Universal Robots PolyScope program: pr1.urp

Program pr1 (installation=default directory=/programs createdIn=5.5.1.82186 lastSavedIn=5.5.1.82186 robotSerialNumber=20195300809)
Calibrated DH parameters: a=[-0.000085, -0.20076, -0.212369, 0.000121, -0.000118, 0]; d=[0.15185, -26.306375, 24.753047, 1.684739, 0.085386, 0.092088]; alpha=[1.572149, -0.00522, -0.011864, 1.571339, -1.571085, 0]; deltaTheta=[0, 0.599885, -0.513355, -0.086555, 0.000006, 0]
BeforeStart
  URCap Gripper (Robotiq_Grippers, Robotiq Inc.) dataModel(position=0.0, force=100.0, speed=100.0, positionInDouble=0.0, forceInDouble=100.0, speedInDouble=100.0, slaveIds=[9], blocking=true)
  MoveJ speed 30 deg/s, acceleration 80 deg/s^2 (useActiveTCP=true) feature=Base
    Waypoint punt1: TCP in base x=-102.832 y=-139.085 z=685.946 mm, rx=-1.1427 ry=-1.3106 rz=1.2216 rad; joints [-11.105, -100.438, 18.426, -96.643, -75.028, -3.585] deg
Robot Program (runOnlyOnce=false)
  MoveJ speed 15 deg/s, acceleration 80 deg/s^2 (useActiveTCP=true) feature=Base
    Waypoint Agafar: TCP in base x=-468.862 y=-44.814 z=176.236 mm, rx=2.2701 ry=1.9757 rz=0.096 rad; joints [-11.109, -45.141, 57.796, -94.518, -89.172, -3.354] deg; TCP offset x=0 y=0 z=0 mm, rx=0 ry=0 rz=0 rad
    URCap Gripper (Robotiq_Grippers, Robotiq Inc.) dataModel(position=100.0, force=100.0, speed=100.0, positionInDouble=100.0, forceInDouble=100.0, speedInDouble=100.0, slaveIds=[9], blocking=true)
  If digital_out[0]≟ True
    MoveJ speed 60 deg/s, acceleration 80 deg/s^2 (useActiveTCP=true) feature=Base
      Waypoint punt1: TCP in base x=-102.832 y=-139.085 z=685.946 mm, rx=-1.1427 ry=-1.3106 rz=1.2216 rad; joints [-11.105, -100.438, 18.426, -96.643, -75.028, -3.585] deg
